FUNCTION_BLOCK PUBLIC FB_PartPresence

VAR_IN_OUT
	HardwareOutputArray : ARRAY [*] OF BOOL; 	// For Sensors
END_VAR

VAR
	Configuration 		: ST_PartPresenceConfiguration;
	Status				: ST_PartPresenceStatus;
	
	InitDone 			: BOOL := FALSE;
	
	OnTimer				: TON;
	OffTimer			: TON;
END_VAR

IF NOT InitDone THEN
	M_Init();
	InitDone:= TRUE;
ELSE
	M_Cyclic();
END_IF

METHOD PRIVATE M_Cyclic : BOOL
VAR_INPUT
END_VAR
IF Configuration.ActivationType = E_ActivationType.NormallyOpen THEN
	OnTimer.IN := Configuration.HardwareInput;
	OnTimer.PT := Configuration.DebounceOnTime;
	
	OffTimer.IN := NOT Configuration.HardwareInput;
	OffTimer.PT := Configuration.DebounceOffTime;
	
ELSIF Configuration.ActivationType = E_ActivationType.NormallyClosed THEN
	OnTimer.IN := NOT Configuration.HardwareInput;
	OnTimer.PT := Configuration.DebounceOnTime;
	
	OffTimer.IN := Configuration.HardwareInput;
	OffTimer.PT := Configuration.DebounceOffTime;
END_IF

OnTimer();
OffTimer();

IF OnTimer.Q THEN
	Status.isOn := TRUE;
ELSIF OffTimer.Q THEN
	Status.isOn := FALSE;
END_IF
END_METHOD

METHOD PRIVATE M_Init : BOOL
VAR_INPUT
END_VAR
END_METHOD

METHOD PUBLIC M_Reset : BOOL
VAR_INPUT
END_VAR
END_METHOD

PROPERTY PUBLIC P_Configuration : REFERENCE TO ST_PartPresenceConfiguration
GET
P_Configuration REF= Configuration;
END_GET
END_PROPERTY

PROPERTY PUBLIC P_Status : REFERENCE TO ST_PartPresenceStatus
GET
P_Status REF= Status;
END_GET
END_PROPERTY

END_FUNCTION_BLOCK

(* stored: Version 1.1.0.1, ProductVersion 3.1.4024.12
   POU FB_PartPresence: Id {91d44c99-a00f-456f-9785-5068ea359f2a}, SpecialFunc None
   Method M_Cyclic: Id {68a0d46e-cd53-4bd0-a175-e664883e7c6d}
   Method M_Init: Id {52915d40-941a-4dcb-b873-76110f25a70f}
   Method M_Reset: Id {b6304d0e-d4d1-434e-a2c0-0221294e00a7}
   Property P_Configuration: Id {40a4ce23-bf31-4469-9096-444c9507dd4b}
   Get Get: Id {b439ea53-4971-465a-83d3-3bf69e1f3812}
   Property P_Status: Id {b44d4190-ebeb-4504-b3ec-016f61130c32}
   Get Get: Id {98c11dca-c0d5-42c3-94aa-155d13475fa7} *)
